% RSLogix 500 project AUBAI_Mixing_tank.RSS, saved by version 8.30.00.16 %
PROJECT "UNTITLED"    % processor: Bul.1763 MicroLogix 1100 Series B %

PROGRAM FILES
  LAD 2   5 rungs

DATA FILES
  O0 OUTPUT  4 elements
  I1 INPUT  6 elements
  S2 STATUS  66 elements
  B3 BINARY  1 elements
  T4 TIMER  2 elements
  C5 COUNTER  1 elements
  R6 CONTROL  1 elements
  N7 INTEGER  1 elements
  F8 FLOAT  1 elements

LADDER 2
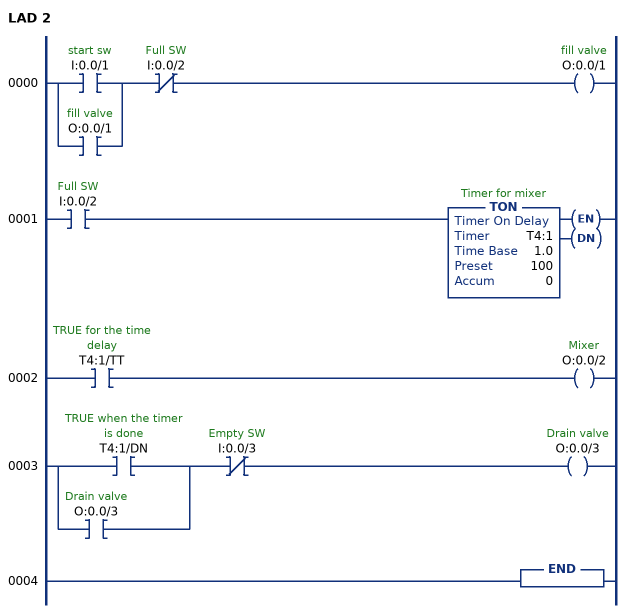
% Rung: 0 %
SOR BST XIC I:0.0/1 NXB XIC O:0.0/1 BND XIO I:0.0/2 OTE O:0.0/1 EOR
%   I:0.0/1  "start sw" %
%   O:0.0/1  "fill valve" %
%   I:0.0/2  "Full SW" %
% Rung: 1 %  % edit flag set %
SOR XIC I:0.0/2 TON T4:1 1.0 100 0 EOR
%   I:0.0/2  "Full SW" %
%   T4:1  "Timer for mixer" %
% Rung: 2 %
SOR XIC T4:1/TT OTE O:0.0/2 EOR
%   T4:1/TT  "TRUE for the time delay" %
%   O:0.0/2  "Mixer" %
% Rung: 3 %
SOR BST XIC T4:1/DN NXB XIC O:0.0/3 BND XIO I:0.0/3 OTE O:0.0/3 EOR
%   T4:1/DN  "TRUE when the timer is done" %
%   O:0.0/3  "Drain valve" %
%   I:0.0/3  "Empty SW" %
% Rung: 4 %
SOR END EOR

OTHER DOCUMENTED ADDRESSES
  I:1.0/0  "Start sw"
  I:1.0/1  "Full sw"
  I:1.0/2  "Empty sw"
  O:2.0/0  "Fill valve"
  O:2.0/1  "Mixer"
  O:2.0/3  "Drain valve"

DATA TABLE (non-zero values as saved)
DATA T4
% .PRE .ACC %
% T4:1 % 1000 0
